// TIA Portal V18 export
// export: Created 2025-12-01T17:51:03.2881134Z, ExportSetting None, DisplayName Totally Integrated Automation Portal, DisplayVersion V18 Update 5, DisplayName TIA Portal Openness, DisplayVersion V18 Update 5, DisplayName TIA Portal Teamcenter Gateway, DisplayVersion V18, DisplayName TIA Portal Version Control Interface, DisplayVersion V18, DisplayName STEP 7 Professional, DisplayVersion V18 Update 5, DisplayName STEP 7 Safety, DisplayVersion V18, DisplayName WinCC Professional, DisplayVersion V18 Update 5
DATA_BLOCK "ST10_CountCycleTimeMain_DB"   // DB1009
// stored: AutoNumber false, InstanceOfName ST10_CountCycleTimeMain, InstanceOfType FB
"ST10_CountCycleTimeMain"
   // VAR_INPUT
   //    iAlwaysOn : Bool;
   //    iRun : Bool;
   //    iManualMode : Bool;
   //    iAutoMode : Bool;
   //    iAutoRunning : Bool;
   // END_VAR
   // VAR
   //    MianCountCycleTime { S7_SetPoint := 'True'} : "Count_CycleTime";
   //    PM1CountCycleTime { S7_SetPoint := 'True'} : "Count_CycleTime_V3";
   //    PM2CountCycleTime { S7_SetPoint := 'True'} : "Count_CycleTime_V3";
   //    PM3CountCycleTime { S7_SetPoint := 'True'} : "Count_CycleTime_V3";
   //    PM4CountCycleTime { S7_SetPoint := 'True'} : "Count_CycleTime_V3";
   //    PM5CountCycleTime { S7_SetPoint := 'True'} : "Count_CycleTime_V3";
   //    PM6CountCycleTime { S7_SetPoint := 'True'} : "Count_CycleTime_V3";
   //    PM7CountCycleTime { S7_SetPoint := 'True'} : "Count_CycleTime_V3";
   //    PM8CountCycleTime { S7_SetPoint := 'True'} : "Count_CycleTime_V3";
   //    PM9CountCycleTime { S7_SetPoint := 'True'} : "Count_CycleTime_V3";
   //    PM10CountCycleTime { S7_SetPoint := 'True'} : "Count_CycleTime_V3";
   //    PM11CountCycleTime { S7_SetPoint := 'True'} : "Count_CycleTime_V3";
   //    PM12CountCycleTime { S7_SetPoint := 'True'} : "Count_CycleTime_V3";
   //    PM13CountCycleTime { S7_SetPoint := 'True'} : "Count_CycleTime_V3";
   //    PM14CountCycleTime { S7_SetPoint := 'True'} : "Count_CycleTime_V3";
   //    PM15CountCycleTime { S7_SetPoint := 'True'} : "Count_CycleTime_V3";
   //    PM16CountCycleTime { S7_SetPoint := 'True'} : "Count_CycleTime_V3";
   //    PM17CountCycleTime { S7_SetPoint := 'True'} : "Count_CycleTime_V3";
   //    PM18CountCycleTime { S7_SetPoint := 'True'} : "Count_CycleTime_V3";
   //    PM19CountCycleTime { S7_SetPoint := 'True'} : "Count_CycleTime_V3";
   //    PM20CountCycleTime { S7_SetPoint := 'True'} : "Count_CycleTime_V3";
   //    PM21CountCycleTime { S7_SetPoint := 'True'} : "Count_CycleTime_V3";
   //    PM22CountCycleTime { S7_SetPoint := 'True'} : "Count_CycleTime_V3";
   //    PM23CountCycleTime { S7_SetPoint := 'True'} : "Count_CycleTime_V3";
   //    PM24CountCycleTime { S7_SetPoint := 'True'} : "Count_CycleTime_V3";
   //    PM25CountCycleTime { S7_SetPoint := 'True'} : "Count_CycleTime_V3";
   //    PM26CountCycleTime { S7_SetPoint := 'True'} : "Count_CycleTime_V3";
   //    PM27CountCycleTime { S7_SetPoint := 'True'} : "Count_CycleTime_V3";
   //    PM28CountCycleTime { S7_SetPoint := 'True'} : "Count_CycleTime_V3";
   //    PM29CountCycleTime { S7_SetPoint := 'True'} : "Count_CycleTime_V3";
   //    PM30CountCycleTime { S7_SetPoint := 'True'} : "Count_CycleTime_V3";
   // END_VAR
BEGIN
END_DATA_BLOCK
